GLOBALCONSTANTS DefaultPool_Dreieck_BargraphSplit (* Split-bargraph constants (left/right object IDs, shared magnitude bounds) *)
  PACKAGE Uebungen::const::UT::Dreieck;
  VAR_GLOBAL CONSTANT
    Bargraph_Split_BargraphSplit : isobus::utils::bargraph::BargraphSplit_S := (stLeft := (u16ObjId := 18001, r32Scale := 1.0, i32Offset := 0, u8Decimals := 0), stRight := (u16ObjId := 18002, r32Scale := 1.0, i32Offset := 0, u8Decimals := 0), r32MinMagnitude := 0.0, r32MaxMagnitude := 42.0);
  END_VAR
END_GLOBALCONSTANTS
